// TIA Portal project "Project1" (V16)

(* hardware
DEVICE "PC-System_1"  SIMATIC PC station
   slot 0: "SIMATIC PC station"  Rail  SIMATIC PC-Station  V1.0
      slot 125: "Stationmanager"  Station_Manager  V6.0.4
   slot 1: "HMI_RT_1"  WinCC RT Advanced  6AV2 104-0xxxx-xxxx  16.0.0.0
      slot 33792: "Computer interface"  Host interface
   slot 2: "IE general_1"  IE General  IE_CP  V8.2.0
*)

(* ===== HMI "HMI_RT_1" =====
system functions are stored by id; their names below are inferred from use
connection "Connection_1": OPC, OPC
connection "Connection_2": OPC, OPC_UA

HMI tags "Default tag table"
   "PV_COUNT_1" : Int, internal
   "PV_COUNT_2" : Int, internal
   "Y" : Int, internal
   "DEN1" : VT_I2 AT Dev01.Tag_Output.Y0, 1 s
   "DEN2" : VT_I2 AT Dev01.Tag_Output.Y1, 1 s
   "DEN3" : VT_I1 AT Dev01.Tag_Output.Y2, 1 s
   "DEN4" : VT_I1 AT Dev01.Tag_Output.Y3, 1 s

HMI tags "Tag table_1"
   "Y1" : VT_BOOL AT Dev01.Tag_Output.Y1, 1 s
   "Y2" : VT_BOOL AT Dev01.Tag_Output.Y2, 1 s
   "Y3" : VT_BOOL AT Dev01.Tag_Output.Y3, 1 s
   "X0" : VT_BOOL AT Dev01.Tag_Input.X0, 1 s
   "X1" : VT_BOOL AT Dev01.Tag_Input.X1, 1 s
   "X2" : VT_BOOL AT Dev01.Tag_Input.X2, 1 s
   "X3" : VT_BOOL AT Dev01.Tag_Input.X3, 1 s
   "X4" : VT_BOOL AT Dev01.Tag_Input.X4, 1 s
   "X5" : VT_BOOL AT Dev01.Tag_Input.X5, 1 s
   "X6" : VT_BOOL AT Dev01.Tag_Input.X6, 1 s
   "X7" : VT_BOOL AT Dev01.Tag_Input.X7, 1 s
   "X8" : VT_BOOL AT Dev01.Tag_Input.X10, 1 s
   "X9" : VT_BOOL AT Dev01.Tag_Input.X11, 1 s
   "Y0" : VT_BOOL AT Dev01.Tag_Output.Y0, 1 s
   "T1" : VT_I2 AT Dev01.Tag_Input.T1_COUNT, 1 s
   "T2" : VT_I2 AT Dev01.Tag_Input.T2_COUNT, 1 s

screen "Log in" 1024x768
   DateTimeField "Date/time field_1" at 778,164 size 212x31
   Clock "Clock_1" at 824,19 size 120x120
   TextField "Text field_15" at 25,308 size 356x22; Text 'Giảng viên hướng dẫn : Ths. Nguyễn Quang Nhã'
   TextField "Text field_16" at 28,342 size 221x22; Text 'Tên người làm: Hoàng Bá Duy'
   TextField "Text field_17" at 268,4 size 449x32; Text 'Hệ thống điều khiển xung mạch cầu H'
   UserView "User view_1" at 544,282 size 480x240
   TextField "Text field_18" at 369,95 size 131x32; Text 'Đăng nhập'
   Button "Button_11" at 389,156 size 96x32; TextOff 'System'; Authorization "Operate"
      on Click: ActivateScreen("Operation", 0)

screen "Operation" 1024x768
   Circle "Circle_1" at 464,128 size 48x48
      Appearance <- "Y0"
   Button "Button_1" at 98,104 size 96x32; TextOff 'START'
      on Release: ResetBit("X0")
      on Press: SetBit("X0")
   Button "Button_2" at 98,145 size 95x27; TextOff 'STOP'
      on Release: ResetBit("X1")
      on Press: SetBit("X1")
   TextField "Text field_1" at 106,70 size 85x22; Text 'Điều khiển'
   IOField "I/O field_1" at 552,327 size 96x32; FormatPattern 9999
      ProcessValue <- "T1"
      Appearance <- "T1"
   Circle "Circle_2" at 625,128 size 48x48
      Appearance <- "Y2"
   Circle "Circle_3" at 464,224 size 48x48
      Appearance <- "Y1"
   Circle "Circle_4" at 625,224 size 48x48
      Appearance <- "Y3"
   Button "Button_3" at 104,261 size 96x32; TextOff 'UNIPOLAR'
      on Release: ResetBit("X4")
      on Press: SetBit("X4")
      Appearance <- "X4"
   Button "Button_4" at 104,304 size 96x32; TextOff 'BIPOLAR'
      on Release: ResetBit("X5")
      on Press: SetBit("X5")
      Appearance <- "X5"
   TextField "Text field_5" at 105,222 size 84x22; Text 'POLARITY'
   TextField "Text field_7" at 546,197 size 33x22; Text 'Vab'
   TextField "Text field_8" at 531,177 size 15x22; Text 'A'
   TextField "Text field_9" at 327,169 size 31x22; Text 'Vcc'
   TextField "Text field_10" at 575,178 size 15x22; Text 'B'
   DateTimeField "Date/time field_1" at 42,397 size 212x31
   TextField "Text field_11" at 345,336 size 207x22; Text 'Thời gian chạy UNIPOLAR:'
   IOField "I/O field_3" at 552,377 size 96x32; FormatPattern 9999
      ProcessValue <- "T2"
   TextField "Text field_12" at 356,381 size 194x22; Text 'Thời gian chạy BIPOLAR:'
   TextField "Text field_13" at 653,329 size 37x22; Text 'giây'
   TextField "Text field_14" at 653,380 size 37x22; Text 'giây'
   Clock "Clock_1" at 824,19 size 120x120
   TextField "Text field_15" at 23,461 size 356x22; Text 'Giảng viên hướng dẫn : Ths. Nguyễn Quang Nhã'
   TextField "Text field_16" at 26,495 size 221x22; Text 'Tên người làm: Hoàng Bá Duy'
   UserView "User view_1" at 544,505 size 480x240
   TextField "Text field_17" at 268,4 size 449x32; Text 'Hệ thống điều khiển xung mạch cầu H'
   Button "Button_11" at 152,613 size 96x32; TextOff 'Sign out'
      on Click: ActivateScreen("Log in", 0)
   Button "Button_12" at 290,612 size 100x35; TextOff 'Show graph'; Authorization "User administration"
      on Click: ActivateScreen("Graph", 0)
   TextField "Text field_18" at 277,574 size 151x22; Text 'Xem log tại C:\Logs'
   TextField "Text field_19" at 191,657 size 286x22; Text '!Note : Chỉ Admin mới được xem graph'
   TextField "Text field_2" at 477,70 size 63x22; Text 'Hiển thị'

screen "Graph" 1024x768
   TrendView "Trend view_1" at 0,0 size 978x614
   Button "Button_1" at 7,620 size 124x32; TextOff 'Back to home'
      on Click: ActivateScreen("Operation", 0)
   Button "Button_2" at 193,619 size 99x33; TextOff 'Sign out'
      on Click: ActivateScreen("Log in", 0)
*)